FUNCTION_BLOCK FB_TcLoggerHandler EXTENDS FB_Handler
VAR_INPUT
END_VAR
VAR_OUTPUT
END_VAR
VAR
END_VAR

SUPER^();

METHOD PUBLIC M_Request
VAR_INPUT
	stEvent:			ST_Event;		// event to be handled. 
END_VAR
VAR
	nFind:				INT;
END_VAR
IF stEvent.bEvent THEN
	CASE stEvent.eEvent OF
		E_Event.Debug:
			ADSLOGSTR(ADSLOG_MSGTYPE_HINT OR ADSLOG_MSGTYPE_LOG, stEvent.sMessage, '');
		E_Event.Info:
			ADSLOGSTR(ADSLOG_MSGTYPE_HINT OR ADSLOG_MSGTYPE_LOG, stEvent.sMessage, '');
		E_Event.Warning:
			ADSLOGSTR(ADSLOG_MSGTYPE_WARN OR ADSLOG_MSGTYPE_LOG, stEvent.sMessage, '');
		E_Event.Error:
			ADSLOGSTR(ADSLOG_MSGTYPE_ERROR OR ADSLOG_MSGTYPE_LOG, stEvent.sMessage, '');
	END_CASE
END_IF

SUPER^.M_Request(stEvent);
END_METHOD

END_FUNCTION_BLOCK

(* stored: Version 1.1.0.1, ProductVersion 3.1.4024.12
   POU FB_TcLoggerHandler: Id {f8a57a06-ef70-4bb8-94fe-c0bb0d78a6cc}, SpecialFunc None
   Method M_Request: Id {adf3dd9b-244f-44a9-8444-44a7adbab493} *)
